{attribute 'qualified_only'}
{attribute 'strict'}
{attribute 'to_string'}
TYPE E_TurntableErrorCode :
(
    None                 := 16#0000,
    InvalidPositionState := 16#7101,
    PositionTimeout      := 16#7102, // 转台绝对定位超时
    InvalidProcessStep   := 16#71FF
) UDINT;
END_TYPE

(* stored: Version 1.1.0.1, ProductVersion 3.1.4026.20
   DUT E_TurntableErrorCode: Id {734eb9ae-66f2-4509-8fbd-99d209d8512f} *)
